// TIA Portal V20 export
TYPE "type_emRelations_em0_cmStatus"
// stored: Access Published, Namespace Unit1
   STRUCT
      cmTopDirectionCheckSensor { S7_SetPoint := 'True'} : "LBC_typeDigitalSignalControlNode";
      cmRadiusMeasureTop { ExternalAccessible := 'False'; ExternalVisible := 'False'; ExternalWritable := 'False'} : "LBC_typeAnalogInputControlNode";
      cmRadiusMeasure { ExternalWritable := 'False'} : "LER_typeRadiusMeasureControlNode";
      cmUnwinderTopAxisB { ExternalAccessible := 'False'; ExternalVisible := 'False'; ExternalWritable := 'False'; S7_SetPoint := 'True'} : "LBC_typeAxis64PosControlNode";
      cmAirShaftTopOnOff { ExternalAccessible := 'False'; ExternalVisible := 'False'; ExternalWritable := 'False'; S7_SetPoint := 'True'} : "LBC_typeTwoWayActuatorControlNode";
      cmEpcTop { ExternalAccessible := 'False'; ExternalVisible := 'False'; ExternalWritable := 'False'} : "LER_typeCON600ControlNode";
   END_STRUCT;
   // cmTopDirectionCheckSensor.commands.reset := FALSE;
   // cmTopDirectionCheckSensor.commands.simulation := FALSE;
   // cmTopDirectionCheckSensor.commands.quality := TRUE;
   // cmRadiusMeasureTop.commands.simulation := FALSE;
   // cmRadiusMeasureTop.commands.reset := FALSE;
   // cmRadiusMeasureTop.commands.quality := TRUE;
   // cmRadiusMeasureTop.monitoring.valid := FALSE;
   // cmRadiusMeasureTop.monitoring.busy := FALSE;
   // cmRadiusMeasureTop.monitoring.error := TRUE;
   // cmRadiusMeasureTop.monitoring.status := 16#8405;
   // cmRadiusMeasureTop.monitoring.processValue := 0.0;
   // cmRadiusMeasureTop.monitoring.limitHigh2 := FALSE;
   // cmRadiusMeasureTop.monitoring.limitHigh1 := FALSE;
   // cmRadiusMeasureTop.monitoring.limitLow1 := FALSE;
   // cmRadiusMeasureTop.monitoring.limitLow2 := FALSE;
   // cmRadiusMeasureTop.monitoring.maxValueReached := FALSE;
   // cmRadiusMeasureTop.monitoring.minValueReached := TRUE;
   // cmRadiusMeasure.commands.ZeroSet := FALSE;
   // cmRadiusMeasure.commands.Reset := FALSE;
   // cmRadiusMeasure.monitoring.Radius := 39.0;
   // cmRadiusMeasure.monitoring.Diameter := 78.0;
END_TYPE
